FUNCTION_BLOCK fbDrive
VAR	
	_position : LREAL;
	_speed : LREAL;
	_acc_dcc : LREAL;
	
	_targetPosition : LREAL;
	_targetSpeed : LREAL;
	_targetAccDcc : LREAL;
END_VAR

METHOD MoveAbsolute : BOOL
VAR_INPUT
	Position : LREAL;
	Speed : LREAL;
	AccDcc : LREAL;
END_VAR
_targetPosition := Position;
_targetSpeed := Speed;
_targetAccDcc := AccDcc;

MoveAbsolute := 
     _targetPosition = Position;
END_METHOD

END_FUNCTION_BLOCK

(* stored: Version 1.1.0.1, ProductVersion 3.1.4024.5
   POU fbDrive: Id {6b100403-3442-4127-b0c9-74cb445ed69a}, SpecialFunc None
   Method MoveAbsolute: Id {ead30145-a48e-4801-b0e4-06d223b0dede} *)
